INTERFACE I_FileEntry EXTENDS I_FileSystemEntry

METHOD GetFullPath : T_MaxString
END_METHOD

PROPERTY Name : T_MaxString
GET
END_GET
SET
END_SET
END_PROPERTY

END_INTERFACE

(* stored: Version 1.1.0.1, ProductVersion 3.1.4024.9
   Itf I_FileEntry: Id {d7cea8c2-6a4b-46b6-9174-113c9c1fd3ed}
   Method GetFullPath: Id {3cfc7bf9-df3b-45bc-8547-790878e96580}
   Property Name: Id {745f4ffb-0dba-459f-be06-2210af6ff534}
   Get Get: Id {a15d2642-d8bc-49c8-8f18-76d76e363704}
   Set Set: Id {0a4169c3-1e37-4f46-97b1-61770d525342} *)
